// TIA Portal V18 export
VAR_GLOBAL   // PLC tag table "02_EL-2"
   "iEL-2p" AT %I0.5 : Bool;
   "iEL-2" AT %I0.6 : Bool;
   "oEL-2p" AT %Q0.0 : Bool;
   "oEL-2" AT %Q0.1 : Bool;
END_VAR
